{attribute 'linkalways'} 
{attribute 'no_explicit_call' := 'This FB is a CLASS and must be accessed using methods or properties'}
{attribute 'enable_dynamic_creation'}
{attribute 'TcRpcEnable'}
FUNCTION_BLOCK AsyncRpcCallQueue IMPLEMENTS I_AsyncRpcCallQueue
VAR
	callQueue : Queue;
END_VAR

METHOD PUBLIC CreateCall : I_AsyncRpcCall
VAR_INPUT
	CallingParameters : I_Deserializer;
	CallingAsynchronousRpcResponse : I_AsynchronousRpcResponse;
	CallingHandler : I_AsynchronousRpcHandler;
END_VAR
VAR
	pAsyncRpcCall : POINTER TO AsyncRpcCall;
END_VAR
pAsyncRpcCall := __NEW(AsyncRpcCall(Parameters := CallingParameters, AsynchronousRpcResponse := CallingAsynchronousRpcResponse, Handler := CallingHandler));
CreateCall := pAsyncRpcCall^;
END_METHOD

METHOD PUBLIC CyclicCall
VAR
	asyncRpcCall : I_AsyncRpcCall;
END_VAR
IF callQueue.TryDequeue(asyncRpcCall) THEN
	asyncRpcCall.Call();
	asyncRpcCall.Dispose();
END_IF
END_METHOD

METHOD PROTECTED DisposeAll
VAR
	asyncRpcCall : I_AsyncRpcCall;
END_VAR
WHILE callQueue.TryDequeue(asyncRpcCall) DO
	asyncRpcCall.Dispose();
END_WHILE
END_METHOD

METHOD FB_exit : BOOL
VAR_INPUT
	bInCopyCode : BOOL; // if TRUE, the exit method is called for exiting an instance that is copied afterwards (online change).
END_VAR
IF bInCopyCode THEN
	RETURN;
END_IF

DisposeAll();
END_METHOD

METHOD PUBLIC TryAddRpcCall : BOOL
VAR_INPUT
	CallingParameters : I_Deserializer;
	CallingAsynchronousRpcResponse : I_AsynchronousRpcResponse;
	CallingHandler : I_AsynchronousRpcHandler;
END_VAR
VAR
	asyncRpcCall : I_AsyncRpcCall;
END_VAR
asyncRpcCall := CreateCall(CallingParameters, CallingAsynchronousRpcResponse, CallingHandler);
callQueue.Enqueue(asyncRpcCall);
TryAddRpcCall := TRUE;
END_METHOD

END_FUNCTION_BLOCK

(* stored: Version 1.1.0.1, ProductVersion 3.1.4024.12
   POU AsyncRpcCallQueue: Id {cccde89e-fed5-416b-8fc0-432729af299f}, SpecialFunc None
   Folder Destructor: Id {cbb8baf2-de67-4823-9b47-93b2cddd1fb5}
   Folder Protected: Id {230bc0d4-752a-4c70-ba9e-5cd3cef4e9b3}
   Method CreateCall: Id {8047f1f6-c70b-40a7-b69a-ac32d2d6fe53}
   Method CyclicCall: Id {162fd676-b57c-4b78-ba17-0fd50a52cb6b}
   Method DisposeAll: Id {dab5ff76-24f9-4911-8300-09993a541f96}
   Method FB_exit: Id {e249dd34-4f22-46ca-a502-e9a8fbd70016}
   Method TryAddRpcCall: Id {e6cf1a26-eeb8-4306-a2a7-0b97adfd4292} *)
